{region '#Template'}
	{attribute 'Version' := '1.2.1.0'}
	{attribute 'Tags' := '"LCID": "1031", "Text": "General, Alarms"'}
	{attribute 'Tags' := '"LCID": "1033", "Text": "General, Alarms"'}
	{attribute 'Using' := '"Type": "Template", "URI": "BA2_Param"'}
	{attribute 'Using' := '"Type": "Template", "URI": "EC_AMEV"'}
	{attribute 'Using' := '"Type": "Template", "URI": "ST_BA_BuildingAlarms"'}
	{attribute 'Description' := '"LCID": "1031", "Text": "Gebäude Alarme"'}
	{attribute 'Description' := '"LCID": "1031", "Text": "Gebäude Alarme"'}
	{attribute 'Description' := '"LCID": "1033", "Text": "Building alarms"'}
{endregion}
FUNCTION_BLOCK FB_BA_BuildingAlarms EXTENDS FB_BA_View
VAR_INPUT CONSTANT
	FireAlert			: FB_BA_BI_IO;                      
	Bgly				: FB_BA_BI_IO;
	CentSwiOff			: FB_BA_BV_Op;
END_VAR	
VAR		
	BuildingAlarms		: FB_BA_RawPublisher;
END_VAR
VAR // added by the converter: edge detectors and wires of the graphical bodies
    _s1 : ST_BA_BuildingAlarms;
END_VAR

SUPER^(); // FB_BA_View
FireAlert(); // FB_BA_BI_IO
Bgly(); // FB_BA_BI_IO
CentSwiOff(); // FB_BA_Bv_OP
// compose _s1 : ST_BA_BuildingAlarms
_s1.bBurglary := Bgly.bPresentValue;
_s1.bFireAlert := FireAlert.bPresentValue;
_s1.bCentralOff := CentSwiOff.bPresentValue;
_s1.bForcedVentilation := FALSE;
_s1.bSmokeExtraction := FALSE;
BuildingAlarms(xData := _s1); // FB_BA_RawPublisher

METHOD FB_init : BOOL
VAR_INPUT
	bInitRetains : BOOL; // if TRUE, the retain variables are initialized (warm start / cold start)
	bInCopyCode : BOOL;  // if TRUE, the instance afterwards gets moved into the copy code (online change)
END_VAR
FireAlert.iParent						:= THIS^;
FireAlert.iLabel						:= LblCmpGeneral.BuildingAlarms_FireAlert;	
FireAlert.sObjectName					:= '{Idx=01}';	
FireAlert.sDeviceType					:= '';
FireAlert.bEnOutOfService				:= FALSE;
FireAlert.ePolarity						:= E_BA_Polarity.eReverse;
FireAlert.sActiveText 					:= txtEvent_On;
FireAlert.sInactiveText 				:= txtEvent_Alert;
FireAlert.nStateChangeCount				:= 0;
FireAlert.nActiveTimeElapsed			:= 0;
FireAlert.nEventClassID					:= EC_ID.NC10;
FireAlert.stTimeDelay.nToNormal			:= BA2_Param.nDefTimeDelay_ToNormal;
FireAlert.stTimeDelay.nToAbnormal		:= BA2_Param.nDefTimeDelay_ToAbnormal;
FireAlert.bAlarmValue					:= TRUE;
FireAlert.bAcknowledgeRm				:= FALSE;	
FireAlert.aEventTransitionText[1]		:= txtEvent_Alert;
FireAlert.aEventTransitionText[2]		:= txtEvent_None;
FireAlert.aEventTransitionText[3]		:= txtEvent_Normal;
FireAlert.bEventDetectionEnable			:= TRUE;
FireAlert.aEventEnable[1]				:= TRUE;			//	to_offnormal
FireAlert.aEventEnable[2]				:= TRUE;			//	to_fault
FireAlert.aEventEnable[3]				:= TRUE;			//	to_normal
FireAlert.eEnPlantLock					:= E_BA_LockPriority.eNoLock;	

Bgly.iParent							:= THIS^;
Bgly.iLabel								:= LblCmpGeneral.BuildingAlarms_Bgly;	
Bgly.sObjectName						:= '{Idx=02}';	
Bgly.sDeviceType						:= '';
Bgly.bEnOutOfService					:= FALSE;
Bgly.ePolarity							:= E_BA_Polarity.eReverse;
Bgly.sActiveText 						:= txtEvent_On;
Bgly.sInactiveText 						:= txtEvent_Alert;
Bgly.nStateChangeCount					:= 0;
Bgly.nActiveTimeElapsed					:= 0;
Bgly.nEventClassID						:= EC_ID.NC10;
Bgly.stTimeDelay.nToNormal				:= BA2_Param.nDefTimeDelay_ToNormal;
Bgly.stTimeDelay.nToAbnormal			:= BA2_Param.nDefTimeDelay_ToAbnormal;
Bgly.bAlarmValue						:= TRUE;
Bgly.bAcknowledgeRm						:= FALSE;	
Bgly.aEventTransitionText[1]			:= txtEvent_Alert;
Bgly.aEventTransitionText[2]			:= txtEvent_None;
Bgly.aEventTransitionText[3]			:= txtEvent_Normal; 
Bgly.bEventDetectionEnable				:= TRUE;
Bgly.aEventEnable[1]					:= TRUE;			//	to_offnormal
Bgly.aEventEnable[2]					:= TRUE;			//	to_fault
Bgly.aEventEnable[3]					:= TRUE;			//	to_normal
Bgly.eEnPlantLock						:= E_BA_LockPriority.eNoLock;	
                       	
CentSwiOff.iParent						:= THIS^;
CentSwiOff.iLabel 						:= LblCmpGeneral.BuildingAlarms_CentSwiOff;	
CentSwiOff.sObjectName					:= '{Idx=01}';
CentSwiOff.sInactiveText				:= txtEvent_Off;
CentSwiOff.sActiveText					:= txtEvent_On;
CentSwiOff.bValueRm						:= FALSE;
CentSwiOff.eToggleMode					:= E_BA_ToggleMode.ePushButton;
END_METHOD

END_FUNCTION_BLOCK

(* stored: Version 1.1.0.1, ProductVersion 3.1.4024.9
   POU FB_BA_BuildingAlarms: Id {c12ab7a9-e8e1-4393-833e-3511e1678564}, SpecialFunc None
   Method FB_init: Id {f5460746-b55f-44b4-b4d4-8e07936e6610} *)
